FUNCTION_BLOCK FB_ConveyorEntry_FBD
VAR_INPUT
END_VAR
VAR_OUTPUT
END_VAR
VAR
	
	timer0_emitter : Tc2_Standard.TP;
	EmitterTrigger : BOOL;
	Timer1 : Tc2_Standard.TON;
	Step_0_Standby : BOOL;
	Step_1 : BOOL;
	Step_2 : BOOL;
	Step_3 : BOOL;
	Step_4 : BOOL;
	Step_5 : BOOL;
	Step_6 : BOOL;
	Step_7 : BOOL;
	Step_10 : BOOL;
	Step_15 : BOOL;
	step_last : BOOL;
	
	condition : BOOL;
	
	Opstart_puls_OS : BOOL;

	
	Initialiser_SQ: BOOL;
END_VAR
VAR_IN_OUT
	control_data : PlantAndCMs.Udt_PlantControl_Mode_1;
	
	control_data_vision : CM_Vision_UDT;
	control_data_Conveyor1 : CM_DO_UDT;
	
	control_data_StopBlade : CM_DO_UDT;
	control_data_emitter : CM_DO_UDT;
END_VAR

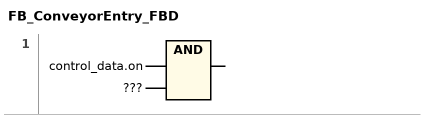
// NETWORK 1
(* control_data.on AND ???; result not used *)

END_FUNCTION_BLOCK

(* stored: Version 1.1.0.1, ProductVersion 3.1.4024.13
   POU FB_ConveyorEntry_FBD: Id {c2840f20-4bb1-436d-bda4-fcbfdcaf086a}, SpecialFunc None *)
